Omron CX-Programmer project NewProject (CX-Programmer 9.03)

# PLC TubesRevisi: CP1L M

## Global symbols (name address type ; comment)
0.00 BOOL  ; START SYSTEM
0.01 BOOL  ; RESET SYSTEM
0.02 BOOL  ; TEMP. CHECKER
0.03 BOOL  ; JALUR AB
0.04 BOOL  ; JALUR AC
0.05 BOOL  ; PROX. A1
0.06 BOOL  ; PROX. B in
0.07 BOOL  ; PROX. B out
0.08 BOOL  ; PROX. A2
0.09 BOOL  ; PROX. C in
0.10 BOOL  ; PROX. C out
0.11 BOOL  ; PROX. A3
100.00 BOOL  ; SYSTEM READY
100.01 BOOL  ; FAILED
100.02 BOOL  ; GOWES
100.03 BOOL  ; RED A
100.04 BOOL  ; GREEN A
100.05 BOOL  ; SERVO
100.06 BOOL  ; GREEN B
100.07 BOOL  ; GREEN C
100.08 BOOL  ; GREEN A
100.09 BOOL  ; PROX. A
100.10 BOOL  ; RED B
100.11 BOOL  ; PROX. B
100.12 BOOL  ; RED C
100.13 BOOL  ; PROX. C
200.00 BOOL  ; VIRTUAL OUTPUT CHECKING
200.01 BOOL  ; VIRTUAL AB
200.02 BOOL  ; VIRTUAL AC
200.03 BOOL  ; VIRTUAL GREEN A
200.04 BOOL  ; VIRTUAL
200.05 BOOL  ; RED B1
200.06 BOOL  ; RED B2
200.07 BOOL  ; GREEN A1
200.08 BOOL  ; GREEN A2
200.09 BOOL  ; RED C1
200.10 BOOL  ; RED C2
200.11 BOOL  ; GREEN A3
D0 CHANNEL  ; COMP. TEMPERATURE
T0000 BOOL  ; GREEN A
T0001 BOOL  ; SERVO (ASUMSI 50 : WAKTU DIBUTUHKAN KERETA MENEMPUH JALUR B)
T0002 BOOL  ; GREEN B
T0003 BOOL  ; RED B
T0004 BOOL  ; GREEN C
T0005 BOOL  ; RED C

## Program NewProgram1 (cyclic task 0)

### Section Section1

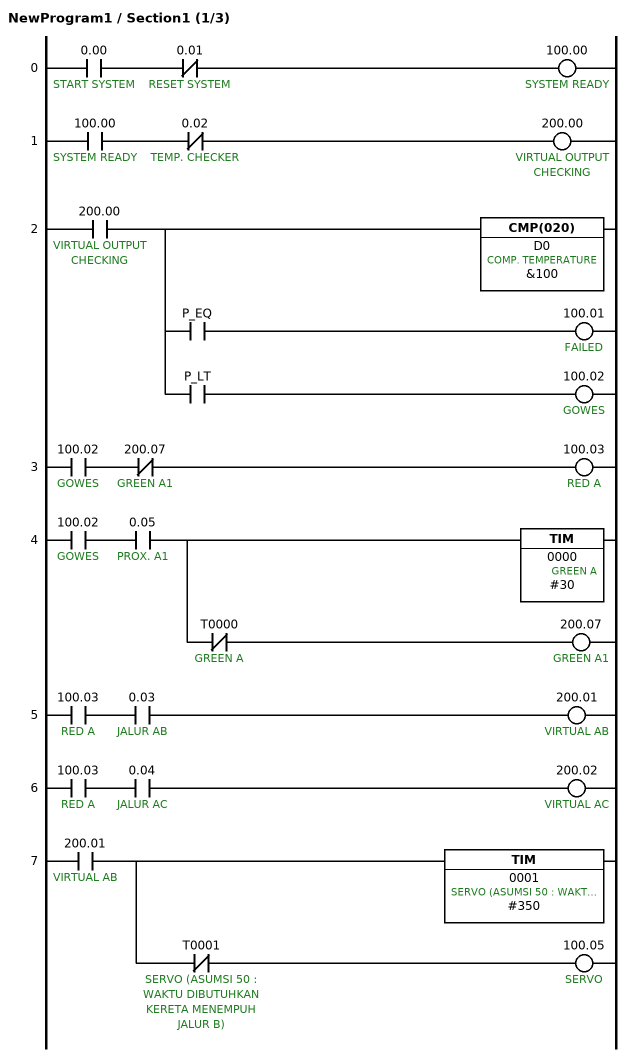
; rung 0
LD 0.00  ; START SYSTEM
ANDNOT 0.01  ; RESET SYSTEM
OUT 100.00  ; SYSTEM READY
; rung 1
LD 100.00  ; SYSTEM READY
ANDNOT 0.02  ; TEMP. CHECKER
OUT 200.00  ; VIRTUAL OUTPUT CHECKING
; rung 2
LD 200.00  ; VIRTUAL OUTPUT CHECKING
OUT TR0
CMP(020) D0 &100  ; COMP. TEMPERATURE
AND P_EQ
OUT 100.01  ; FAILED
LD TR0
AND P_LT
OUT 100.02  ; GOWES
; rung 3
LD 100.02  ; GOWES
ANDNOT 200.07  ; GREEN A1
OUT 100.03  ; RED A
; rung 4
LD 100.02  ; GOWES
AND 0.05  ; PROX. A1
TIM 0000 #30  ; GREEN A
ANDNOT T0000  ; GREEN A
OUT 200.07  ; GREEN A1
; rung 5
LD 100.03  ; RED A
AND 0.03  ; JALUR AB
OUT 200.01  ; VIRTUAL AB
; rung 6
LD 100.03  ; RED A
AND 0.04  ; JALUR AC
OUT 200.02  ; VIRTUAL AC
; rung 7
LD 200.01  ; VIRTUAL AB
TIM 0001 #350  ; SERVO (ASUMSI 50 : WAKTU DIBUTUHKAN KERETA MENEMPUH JALUR B)
ANDNOT T0001  ; SERVO (ASUMSI 50 : WAKTU DIBUTUHKAN KERETA MENEMPUH JALUR B)
OUT 100.05  ; SERVO

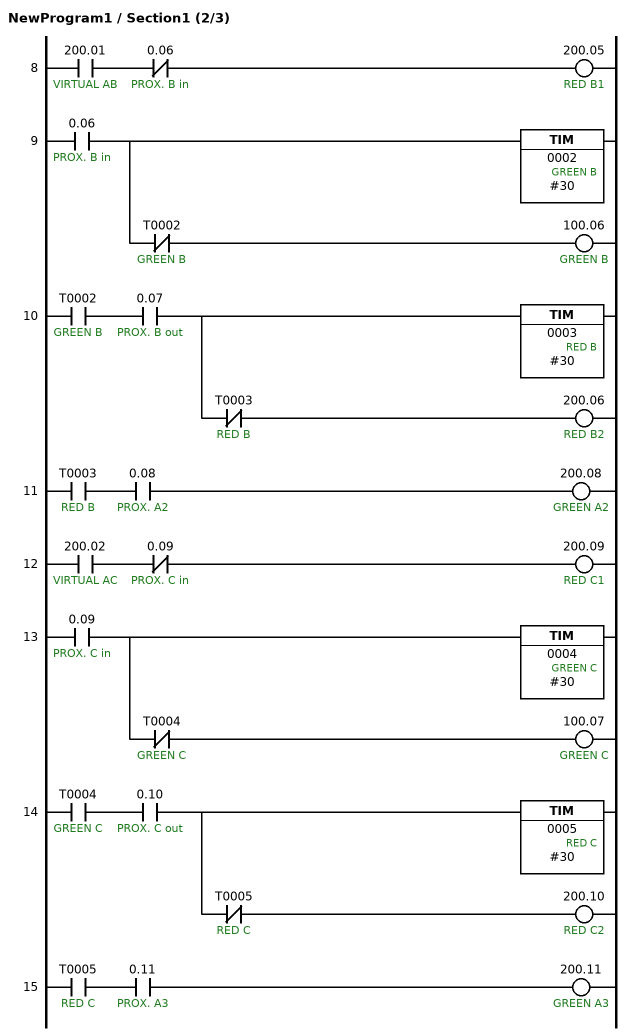
; rung 8
LD 200.01  ; VIRTUAL AB
ANDNOT 0.06  ; PROX. B in
OUT 200.05  ; RED B1
; rung 9
LD 0.06  ; PROX. B in
TIM 0002 #30  ; GREEN B
ANDNOT T0002  ; GREEN B
OUT 100.06  ; GREEN B
; rung 10
LD T0002  ; GREEN B
AND 0.07  ; PROX. B out
TIM 0003 #30  ; RED B
ANDNOT T0003  ; RED B
OUT 200.06  ; RED B2
; rung 11
LD T0003  ; RED B
AND 0.08  ; PROX. A2
OUT 200.08  ; GREEN A2
; rung 12
LD 200.02  ; VIRTUAL AC
ANDNOT 0.09  ; PROX. C in
OUT 200.09  ; RED C1
; rung 13
LD 0.09  ; PROX. C in
TIM 0004 #30  ; GREEN C
ANDNOT T0004  ; GREEN C
OUT 100.07  ; GREEN C
; rung 14
LD T0004  ; GREEN C
AND 0.10  ; PROX. C out
TIM 0005 #30  ; RED C
ANDNOT T0005  ; RED C
OUT 200.10  ; RED C2
; rung 15
LD T0005  ; RED C
AND 0.11  ; PROX. A3
OUT 200.11  ; GREEN A3

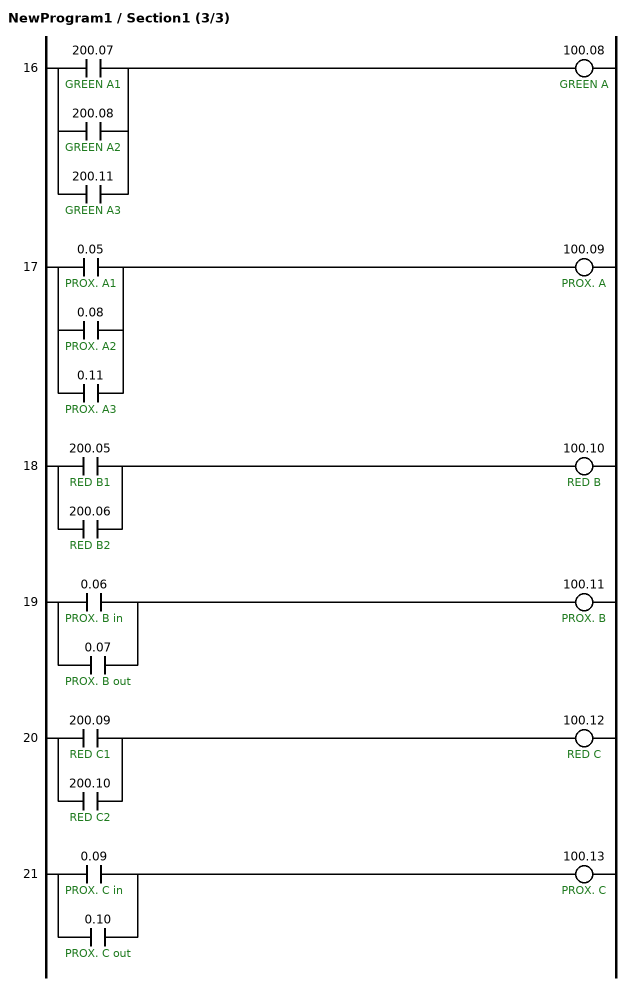
; rung 16
LD 200.07  ; GREEN A1
OR 200.08  ; GREEN A2
OR 200.11  ; GREEN A3
OUT 100.08  ; GREEN A
; rung 17
LD 0.05  ; PROX. A1
OR 0.08  ; PROX. A2
OR 0.11  ; PROX. A3
OUT 100.09  ; PROX. A
; rung 18
LD 200.05  ; RED B1
OR 200.06  ; RED B2
OUT 100.10  ; RED B
; rung 19
LD 0.06  ; PROX. B in
OR 0.07  ; PROX. B out
OUT 100.11  ; PROX. B
; rung 20
LD 200.09  ; RED C1
OR 200.10  ; RED C2
OUT 100.12  ; RED C
; rung 21
LD 0.09  ; PROX. C in
OR 0.10  ; PROX. C out
OUT 100.13  ; PROX. C

### Section END
; rung 0
END(001)